PROGRAM MAIN
VAR
	st_event: ST_Event; // Only this structs copy is being used everywhere.
	once: BOOL := FALSE;
	
	csvEventStorage: FB_CSVEventStorage;
	eventLogger : FB_EventLogger(csvEventStorage);
END_VAR

IF once THEN
	st_event.eEventType := E_EventType.alarm;
	st_event.eEventSeverity := TcEventSeverity.Critical;
	st_event.sEventText :=  'This is an event text';
	
	eventLogger.AddEvent(st_event);
	once := FALSE;
END_IF

csvEventStorage();

(*IF NOT once THEN
	F_UpdateEventTimeStamp(st_event:= st_event);
	once := TRUE;
END_IF
*)

END_PROGRAM

(* stored: Version 1.1.0.1, ProductVersion 3.1.4024.12
   POU MAIN: Id {16dd2937-1a56-496b-9281-972e8d7713a8}, SpecialFunc None *)
